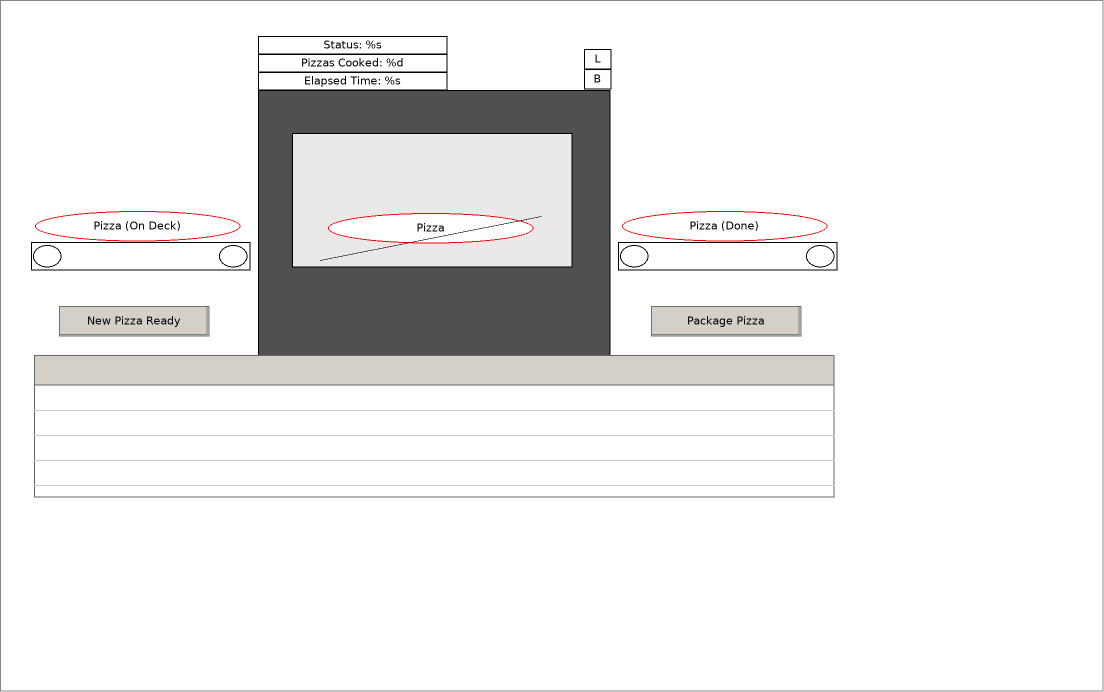
VISUALIZATION Visualization  // 1104x692
    Line (1103,691)
    Rectangle (258,90 352x366)
    Button (59,306 150x30), "New Pizza Ready"
        tap MAIN.bLoadPizza
    Button (651,306 150x30), "Package Pizza"
        tap MAIN.bRemovePizza
    Rectangle (292,133 280x134)
    Ellipse (328,213 205x30), "Pizza", invisible if: NOT MAIN.fbMyPizzaOven[0].stPizzaInOven.bExist
    Rectangle (258,72 189x18), "Elapsed Time: %s", text variable: Main.fbMyPizzaOven[0].fbMyTimer.ET
    Line (320,260) (541,216)
    Rectangle (258,54 189x18), "Pizzas Cooked: %d", text variable: MAIN.fbMyPizzaOven[0].iTotalPizzasCooked
    RoundedRectangle (584,69 27x20), "B", colour toggle: Main.fbMyPizzaOven[0].bBuzzer
    RoundedRectangle (584,49 27x20), "L"
    Rectangle (31,242 219x28)
    Ellipse (35,211 205x30), "Pizza (On Deck)", invisible if: NOT Main.fbMyPizzaOven[0].stPizzaOnDeck.bExist
    Ellipse (33,245 28x22)
    Ellipse (219,245 28x22)
    Rectangle (618,242 219x28)
    Ellipse (622,211 205x30), "Pizza (Done)", invisible if: NOT Main.fbMyPizzaOven[0].stPizzaDone.bExist
    Ellipse (620,245 28x22)
    Ellipse (806,245 28x22)
    Rectangle (258,36 189x18), "Status: %s", text variable: MAIN.fbMyPizzaOven[0].sStateDesc
    Table (34,355 800x142), data array: HMI_VARS.arrPizzaHistory
        p3854506369: HMI_VARS.arrPizzaHistory[INDEX].bExist
        p1892666644: HMI_VARS.arrPizzaHistory[INDEX].dtTimeEnteredOven
        p338671338: HMI_VARS.arrPizzaHistory[INDEX].dtTimeExitedOven
        p2170511999: HMI_VARS.arrPizzaHistory[INDEX].tTimeInOven
        p3723444502: HMI_VARS.arrPizzaHistory[INDEX].eType
END_VISUALIZATION

(* stored: Version 1.1.0.1, ProductVersion 3.1.4024.12
   Visu Visualization: Id {14fe0e48-4827-48e5-b72e-1c1617256d0a} *)
